# B&R Automation Studio project A2019059_Linka_Power_CP (part 43)

#### OvlServaZdvihu.st
```iecst
ACTION OvlServaZdvihu:

	//**************************Axis 11***********************************//
	//Otáčka serva = 10mm//
	//Motor má absolútny encodér a brzdu//

    //ENABLE knižnice//
    IF P4_Etiketovacka.ServoZdvihuEtiketovania_M28.STATUS.Communication_READY THEN
        P4_Etiketovacka.ServoZdvihuEtiketovania_M28.CMD.ENABLE:= TRUE;
    ELSE
        P4_Etiketovacka.ServoZdvihuEtiketovania_M28.CMD.ENABLE:= FALSE;
    END_IF

	//Zapnutie serva//
	CasPowerON.IN:= P4_Etiketovacka.ServoZdvihuEtiketovania_M28.STATUS.ReadyToPower_ON AND P4_Etiketovacka.STAV.ServoZvihu_LimitSnimace_BUSY AND P4_Etiketovacka.ServoZdvihuEtiketovania_M28.STATUS.EnableSwitch_ACTIVE AND NOT P4_Etiketovacka.ServoZdvihuEtiketovania_M28.STATUS.ERROR;
	IF CasPowerON.Q THEN
		P4_Etiketovacka.ServoZdvihuEtiketovania_M28.CMD.POWER:= TRUE;
	ELSE
		P4_Etiketovacka.ServoZdvihuEtiketovania_M28.CMD.POWER:= FALSE;
	END_IF

	CasPowerON.PT:= T#1s;
	CasPowerON();

    //Zobrazenie stavou a parametrov serva//
    P4_Etiketovacka.STAV.Zdvih_AktualnaPozicia:= P4_Etiketovacka.ServoZdvihuEtiketovania_M28.STATUS.ActualPosition;
	P4_Etiketovacka.STAV.Zdvih_AktualnaRychlost:= P4_Etiketovacka.ServoZdvihuEtiketovania_M28.STATUS.ActualVelocity;
	P4_Etiketovacka.STAV.Zdvih_AktualnyMoment:= P4_Etiketovacka.ServoZdvihuEtiketovania_M28.STATUS.ActualTorque;
	P4_Etiketovacka.STAV.ServoZdvihu_HomingOK:= P4_Etiketovacka.ServoZdvihuEtiketovania_M28.STATUS.Homing_OK;
	P4_Etiketovacka.STAV.ServoZdvihu_BUSY:= P4_Etiketovacka.ServoZdvihuEtiketovania_M28.STATUS.MoveAbsolute_BUSY;
	P4_Etiketovacka.STAV.Zdvih_JoggLimitDosiahnuty:= P4_Etiketovacka.ServoZdvihuEtiketovania_M28.STATUS.JoggLimit_Dosiahnuty;

	//Zadané parametre serva//
	P4_Etiketovacka.ServoZdvihuEtiketovania_M28.HomePAR.Acceleration:= 100;
	P4_Etiketovacka.ServoZdvihuEtiketovania_M28.HomePAR.HomingVelocity:= 5;
	P4_Etiketovacka.ServoZdvihuEtiketovania_M28.HomePAR.StartVelocity:= 10;
	P4_Etiketovacka.ServoZdvihuEtiketovania_M28.HomePAR.Position:= -21423.0;    //Offset homing pozície pre absolutny snímač
	P4_Etiketovacka.ServoZdvihuEtiketovania_M28.HomePAR.HomingMode:= 3; //0 - direct, 1- refrenčný snímač, 2 - limitný snímač, 3 - absolutny encoder, 4 - na moment//

	P4_Etiketovacka.ServoZdvihuEtiketovania_M28.PAR.Acceleration:= P34_RemPremenne.P4_ZdvihEtiketovacky_Rychlost*10;
	P4_Etiketovacka.ServoZdvihuEtiketovania_M28.PAR.Deceleration:= P34_RemPremenne.P4_ZdvihEtiketovacky_Rychlost*10;
	P4_Etiketovacka.ServoZdvihuEtiketovania_M28.PAR.StopDeceleration:= P34_RemPremenne.P4_ZdvihEtiketovacky_Rychlost*10;
	P4_Etiketovacka.ServoZdvihuEtiketovania_M28.PAR.Velocity:= P34_RemPremenne.P4_ZdvihEtiketovacky_Rychlost;
	P4_Etiketovacka.ServoZdvihuEtiketovania_M28.PAR.Position:= P4_Etiketovacka.PAR.ServoZdvihu_ZadanaPozicia;

	//Zastavenie pohybu serva//
	IF Zdvih_STOP THEN
		P4_Etiketovacka.ServoZdvihuEtiketovania_M28.CMD.STOP:= TRUE;
		SC_OvlZdvihu.Step:= 0;
		CasZastaveniaServa.IN:= TRUE;
		Zdvih_STOP:= FALSE;
	END_IF

	IF CasZastaveniaServa.Q THEN
		P4_Etiketovacka.ServoZdvihuEtiketovania_M28.CMD.STOP:= FALSE;
		CasZastaveniaServa.IN:= FALSE;
	END_IF

	CasZastaveniaServa.PT:= T#2s;
	CasZastaveniaServa();

	//Volanie funkcie SequenceControl//
	SequenceControl(SC:= SC_OvlZdvihu);

	CASE SC_OvlZdvihu.Step OF

		0:
			SC_OvlZdvihu.StepName:= '0 - Nulovanie';
			Zdvih_JoggHORE:= FALSE;
			Zdvih_JoggDOLE:= FALSE;
			Zdvih_POLOHUJ:= FALSE;
			Zdvih_HOME:= FALSE;
			P4_Etiketovacka.ServoZdvihuEtiketovania_M28.CMD.HOME:= FALSE;
			P4_Etiketovacka.ServoZdvihuEtiketovania_M28.CMD.JoggVPRED:= FALSE;
			P4_Etiketovacka.ServoZdvihuEtiketovania_M28.CMD.JoggVZAD:= FALSE;
			P4_Etiketovacka.ServoZdvihuEtiketovania_M28.CMD.MoveAbsolute:= FALSE;
			P4_Etiketovacka.ServoZdvihuEtiketovania_M28.CMD.MoveTorque:= FALSE;

			IF SC_P4_Etiketovacka.Step <> 0 AND P4_Etiketovacka.ServoZdvihuEtiketovania_M28.STATUS.Power_ON AND NOT P4_Etiketovacka.ServoZdvihuEtiketovania_M28.STATUS.ERROR AND NOT P4_Etiketovacka.ServoZdvihuEtiketovania_M28.STATUS.STOP_ACTIVE THEN
				SC_OvlZdvihu.ResetStep:= TRUE;
				SC_OvlZdvihu.Step:= 1;
			END_IF

		1:
			SC_OvlZdvihu.StepName:= '1 - Rozhodnutie o cinnosti';
			IF Zdvih_JoggHORE THEN
				SC_OvlZdvihu.Step:= 10;
			ELSIF Zdvih_JoggDOLE THEN
				SC_OvlZdvihu.Step:= 20;
			ELSIF Zdvih_HOME THEN
				SC_OvlZdvihu.Step:= 30;
			ELSIF Zdvih_POLOHUJ THEN
				SC_OvlZdvihu.Step:= 40;
			END_IF

		10:
			SC_OvlZdvihu.StepName:= '10 - Jogg HORE';
			SC_OvlZdvihu.IdleTime.PT:= T#3s;
			SC_OvlZdvihu.AlarmTime.PT:= T#3s;

			IF NOT SC_OvlZdvihu.Switch1 THEN
				P4_Etiketovacka.ServoZdvihuEtiketovania_M28.CMD.JoggVZAD:= TRUE;
				SC_OvlZdvihu.Switch1:= TRUE;
			END_IF

			IF NOT Zdvih_JoggHORE THEN
				SC_OvlZdvihu.ResetStep:= TRUE;
				SC_OvlZdvihu.Step:= 0;
			END_IF

		20:
			SC_OvlZdvihu.StepName:= '20 - Jogg DOLE';
			SC_OvlZdvihu.IdleTime.PT:= T#3s;
			SC_OvlZdvihu.AlarmTime.PT:= T#3s;

			IF NOT SC_OvlZdvihu.Switch1 THEN
				P4_Etiketovacka.ServoZdvihuEtiketovania_M28.CMD.JoggVPRED:= TRUE;
				SC_OvlZdvihu.Switch1:= TRUE;
			END_IF

			IF NOT Zdvih_JoggDOLE THEN
				SC_OvlZdvihu.ResetStep:= TRUE;
				SC_OvlZdvihu.Step:= 0;
			END_IF

		30:
			SC_OvlZdvihu.StepName:= '30 - Homing';
			SC_OvlZdvihu.IdleTime.PT:= T#500ms;
			SC_OvlZdvihu.AlarmTime.PT:= T#3s;

			IF NOT SC_OvlZdvihu.Switch1 THEN
				P4_Etiketovacka.ServoZdvihuEtiketovania_M28.CMD.HOME:= TRUE;
				SC_OvlZdvihu.IdleTime.IN:= TRUE;
				SC_OvlZdvihu.Switch1:= TRUE;
			END_IF

			IF P4_Etiketovacka.ServoZdvihuEtiketovania_M28.STATUS.Homing_OK AND SC_OvlZdvihu.IdleTime.Q THEN
				SC_OvlZdvihu.ResetStep:= TRUE;
				SC_OvlZdvihu.Step:= 0;
			END_IF

		40:
			SC_OvlZdvihu.StepName:= '40 - Polohovanie';
			SC_OvlZdvihu.IdleTime.PT:= T#500ms;
			SC_OvlZdvihu.AlarmTime.PT:= T#3s;

			ZadanaPoziciaUINT:= LREAL_TO_UINT(P4_Etiketovacka.PAR.ServoZdvihu_ZadanaPozicia);
			AktualnaPoziciaUINT:= LREAL_TO_UINT(P4_Etiketovacka.STAV.Zdvih_AktualnaPozicia);

			IF NOT SC_OvlZdvihu.Switch1 THEN
				P4_Etiketovacka.ServoZdvihuEtiketovania_M28.CMD.MoveAbsolute:= TRUE;
				SC_OvlZdvihu.Switch1:= TRUE;
			END_IF

			IF (AktualnaPoziciaUINT = ZadanaPoziciaUINT) AND P4_Etiketovacka.ServoZdvihuEtiketovania_M28.STATUS.MoveAbsolute_DONE THEN
				P4_Etiketovacka.STAV.ServoZdvihu_PoziciaDosiahnuta:= TRUE;
				SC_OvlZdvihu.ResetStep:= TRUE;
				SC_OvlZdvihu.Step:= 0;
			END_IF

	END_CASE

END_ACTION
```

#### KOM_Tlaciaren.st
```iecst
ACTION KOM_Tlaciaren:

	CASE Client.sStep OF

		0://Čakanie na spustenie komunikácie z tlačiarňou//
			IF Tlaciaren.Commands.VytlacEtiketu THEN
				Tlaciaren.Status.PoruchaOtvoreniaKomunikacie:= FALSE;
				Tlaciaren.Status.PoruchaSpojenia_s_Tlaciarnou:= FALSE;
				Tlaciaren.Status.PoruchaOdoslaniaDat:= FALSE;
				Tlaciaren.Status.PoruchaZatvoreniaKomunikacie:= FALSE;
				Tlaciaren.Status.PoruchaPrijatiaDat:= FALSE;
				Tlaciaren.Status.PrislaSprava_s_Tlaciarne:= FALSE;
				Tlaciaren.Status.VytlacenieEtikety_ERROR:= FALSE;
				(*strcpy(ADR(Tlaciaren.Data.Sprava_pre_Tlaciaren),ADR(''));*)
				strcpy(ADR(Tlaciaren.Data.Odpoved_s_Tlaciarne),ADR('')); //Vynulovanie premennej typu string
				Client.sStep := 1;
			END_IF

		1: //Otvorenie ethernetovej komunikácie//
			Client.TcpOpen_0.enable := 1;
			Client.TcpOpen_0.pIfAddr := 0;  (* Which Interface to open *)
			Client.TcpOpen_0.port := 9100;  (* Port komunikácie s tlačiarňou *)
			Client.TcpOpen_0.options := 0;
			Client.TcpOpen_0;  (* Call the Function *)

			IF Client.TcpOpen_0.status = 0 THEN  (* TCP port je otvorený *)
				Client.TcpOpen_timeout := 0;
				Client.sStep := 5;
			ELSIF Client.TcpOpen_0.status = ERR_FUB_BUSY THEN  (* TCP port sa otvára *)
				Client.TcpOpen_timeout := Client.TcpOpen_timeout + 1;
				IF Client.TcpOpen_timeout > 50 THEN
					Tlaciaren.Status.PoruchaOtvoreniaKomunikacie:= TRUE;
					Client.TcpOpen_timeout := 0;
					Client.sStep := 40;
				END_IF
				(* Busy *)
			ELSE  (* Goto Error Step *)
				Tlaciaren.Status.PoruchaOtvoreniaKomunikacie:= TRUE;
				Client.TcpOpen_timeout := 0;
				Tlaciaren.Status.VytlacenieEtikety_ERROR:= TRUE;
				Client.sStep := 100;
			END_IF

		5:
			Client.linger_opt.lLinger := 0; (* linger Time = 0 *)
			Client.linger_opt.lOnOff := 1; (* linger Option ON *)
			Client.TcpIoctl_0.enable := 1;
			Client.TcpIoctl_0.ident := Client.TcpOpen_0.ident; (* Connection Ident from AsTP.TCP_Open *)
			Client.TcpIoctl_0.ioctl := tcpSO_LINGER_SET; (* Set Linger Options *)
			Client.TcpIoctl_0.pData := ADR(Client.linger_opt);
			Client.TcpIoctl_0.datalen := SIZEOF(Client.linger_opt);
			Client.TcpIoctl_0;

			IF Client.TcpIoctl_0.status = 0 THEN  (* TcpIoctl successfull *)
				Client.sStep := 10;
			ELSIF Client.TcpIoctl_0.status = ERR_FUB_BUSY THEN  (* TcpIoctl not finished -> redo *)
				(* Busy *)
			ELSE  (* Goto Error Step *)
				Tlaciaren.Status.VytlacenieEtikety_ERROR:= TRUE;
				Client.sStep := 100;
			END_IF

		10: //Spojenie s tlačiarňou//
			Client.TcpClient_0.enable := 1;
			Client.TcpClient_0.ident := Client.TcpOpen_0.ident;  (* Connection Ident from AsTCP.TCP_Open *)
			Client.TcpClient_0.portserv := 9100;  (* Port komunikácie s tlačiarňou *)
			Client.TcpClient_0.pServer := ADR('192.168.122.41');  (* Adresa tlačiarne *)
			Client.TcpClient_0;  (* Call the Function*)

			IF Client.TcpClient_0.status = 0 THEN  (* Open ok -> Send Data *)
				Client.TcpClient_timeout := 0;
				Client.sStep := 20;
			ELSIF Client.TcpClient_0.status = ERR_FUB_BUSY THEN  (* TcpClient not finished -> redo *)
				Client.TcpClient_timeout := Client.TcpClient_timeout + 1;
				IF Client.TcpClient_timeout > 50 THEN
					Tlaciaren.Status.PoruchaSpojenia_s_Tlaciarnou:= TRUE;
					Client.TcpClient_timeout := 0;
					Client.sStep := 40;
				END_IF

				(* Busy *)
			ELSIF Client.TcpClient_0.status = tcpERR_INVALID THEN  (* Port error -> Close actual connection, and reopen a new one *)
				Client.TcpClient_timeout := 0;
				Client.sStep := 40;
			ELSE  (* Goto Error Step *)
				Tlaciaren.Status.PoruchaSpojenia_s_Tlaciarnou:= TRUE;
				Client.TcpClient_timeout := 0;
				Tlaciaren.Status.VytlacenieEtikety_ERROR:= TRUE;
				Client.sStep := 100;
			END_IF

		20: //Poslanie dát do tlačiarne//
			Client.TcpSend_0.enable := 1;
			Client.TcpSend_0.ident := Client.TcpOpen_0.ident;  (* Connection Ident from AsTCP.TCP_Open *)
			Client.TcpSend_0.pData := ADR(Tlaciaren.Data.Sprava_pre_Tlaciaren);  (* Dáta poslané do tlačiarne *)
			Client.TcpSend_0.datalen := SIZEOF(Tlaciaren.Data.Sprava_pre_Tlaciaren);  (* Lenght of data to send *)
			Client.TcpSend_0.flags := 0;
			Client.TcpSend_0;  (* Call the Function*)

			IF Client.TcpSend_0.status = 0 THEN  (* Data was sent sucessfully -> receive data *)
				Client.sStep := 40;
			ELSIF Client.TcpSend_0.status = ERR_FUB_BUSY THEN  (* TcpSend not finished -> redo *)
				(* Busy *)
			ELSIF (Client.TcpSend_0.status = tcpERR_SENTLEN) OR (Client.TcpSend_0.status = tcpERR_NOT_CONNECTED) THEN (* Connection Lost *)
				Client.sStep := 40;
			ELSE  (* Goto Error Step *)
				Tlaciaren.Status.PoruchaOdoslaniaDat:= TRUE;
				Tlaciaren.Status.VytlacenieEtikety_ERROR:= TRUE;
				Client.sStep := 100;
			END_IF

		30: //Prijatie odpovede s tlačiarne//
			Client.TcpRecv_0.enable := 1;
			Client.TcpRecv_0.ident := Client.TcpOpen_0.ident;  (* Connection Ident from AsTCP.TCP_Open *)
			Client.TcpRecv_0.pData	:= ADR(Tlaciaren.Data.Odpoved_s_Tlaciarne);  (* Dáta poslané z tlačiarne *)
			Client.TcpRecv_0.datamax := SIZEOF(Tlaciaren.Data.Odpoved_s_Tlaciarne);  (* Lenght of data buffer *)
			Client.TcpRecv_0.flags := 0;
			Client.TcpRecv_0;  (* Call the Function*)

			IF Client.TcpRecv_0.status = 0 THEN  (* Data was received sucessfully -> Send next packet *)
				Tlaciaren.Status.PrislaSprava_s_Tlaciarne:= TRUE;
				Client.recv_timeout := 0;
				Client.sStep := 40;
			ELSIF Client.TcpRecv_0.status = tcpERR_NO_DATA THEN  (* No data received - wait *)
				Client.recv_timeout := Client.recv_timeout + 1;
				IF Client.recv_timeout > 50 THEN
					Client.recv_timeout := 0;
					Client.sStep := 40;
				END_IF
				(* No Data received *)
			ELSIF Client.TcpRecv_0.status = ERR_FUB_BUSY THEN  (* TcpRecv not finished -> redo *)
				(* Busy *)
			ELSIF Client.TcpRecv_0.status = tcpERR_NOT_CONNECTED THEN (* Connection Lost *)
				Client.recv_timeout := 0;
				Client.sStep := 40;
			ELSE  (* Goto Error Step *)
				Tlaciaren.Status.PoruchaPrijatiaDat:= TRUE;
				Tlaciaren.Status.VytlacenieEtikety_ERROR:= TRUE;
				Client.recv_timeout := 0;
				Client.sStep := 100;
			END_IF

		40: //Zatvorenie ethernetovej komunikácie//
			Client.TcpClose_0.enable := 1;
			Client.TcpClose_0.ident := Client.TcpOpen_0.ident;  (* Connection Ident from AsTCP.TCP_Open *)
			Client.TcpClose_0.how := 0;
			Client.TcpClose_0;  (* Call the Function*)

			IF Client.TcpClose_0.status = 0 THEN  (* Close sucessfull -> Reopen the interface *)
				Tlaciaren.Status.VytlacenieEtikety_OK:= TRUE;
				Client.sStep := 100;
			ELSIF Client.TcpClose_0.status = ERR_FUB_BUSY THEN  (* TcpClose not finished -> redo *)
				(* Busy *)
			ELSE  (* Goto Error Step *)
				Tlaciaren.Status.PoruchaZatvoreniaKomunikacie:= TRUE;
				Tlaciaren.Status.VytlacenieEtikety_ERROR:= TRUE;
				Client.sStep := 100;
			END_IF

		100: //Ukončenie komunikácie s tlačiarňou//
			IF NOT Tlaciaren.Commands.VytlacEtiketu THEN
				Client.sStep := 0;
			END_IF

	END_CASE

END_ACTION
```

#### VytvorenieEtikety.st
```iecst
ACTION VytvorenieEtikety:

	//*********************************************Vyčítanie parametrov etikety zo servera*******************************************************//
	SerioveCisloEtikety;
	IF P4_Etiketovacka.RR_TestovanieEtiketovania THEN
		SerioveCisloEtikety:= 'T598454420120P32120001323091112';
	END_IF

	brsstrcpy(ADR(VstupnePoleUSINT),ADR(SerioveCisloEtikety)); //Skopirovanie vstupnej spravy do pola

    //***************************Vyčítanie Location Code*******************************************//
    brsmemcpy(ADR(Etiketa.LocationCode),ADR(VstupnePoleUSINT[1]),2);

    //**************************Vyčítanie Part Ident Number****************************************//
    brsmemcpy(ADR(Etiketa.PartIdentNumber),ADR(VstupnePoleUSINT[3]),7);

    //**************************Vyčítanie Change Index*********************************************//
    brsmemcpy(ADR(Etiketa.ChangeIndex),ADR(VstupnePoleUSINT[10]),2);

    //**************************Vyčítanie Production Year*********************************************//
    brsmemcpy(ADR(Etiketa.ProductionYear),ADR(VstupnePoleUSINT[12]),2);

    //**************************Vyčítanie Manufactured*********************************************//
    brsmemcpy(ADR(Etiketa.Manufactured),ADR(VstupnePoleUSINT[14]),1);

    //**************************Vyčítanie Day of production*********************************************//
    brsmemcpy(ADR(Etiketa.DayOfProduction),ADR(VstupnePoleUSINT[15]),3);

    //**************************Vyčítanie Assembly line*********************************************//
    brsmemcpy(ADR(Etiketa.AssemblyLine),ADR(VstupnePoleUSINT[18]),1);

    //**************************Vyčítanie Day production counter*********************************************//
    brsmemcpy(ADR(Etiketa.DayProductionCounter),ADR(VstupnePoleUSINT[19]),5);

    //**************************Vyčítanie Supplier number*********************************************//
    brsmemcpy(ADR(Etiketa.SuplierNumber),ADR(VstupnePoleUSINT[24]),6);

    //**************************Vyčítanie Supplier plant code*********************************************//
    brsmemcpy(ADR(Etiketa.PlantCode),ADR(VstupnePoleUSINT[30]),2);

    //*****************************************************Namapovanie parametrov etikety************************************************//

    //Identification number//
    EtiketaPanasonic.IdentificationNumber:= Etiketa.PartIdentNumber;

    //Change Index//
    EtiketaPanasonic.ChangeIndex:= '';
    strcat(ADR(EtiketaPanasonic.ChangeIndex),ADR('-'));
    strcat(ADR(EtiketaPanasonic.ChangeIndex),ADR(Etiketa.ChangeIndex));

    //Model type//
    EtiketaPanasonic.ModelType:= 'POWER-CP';

    //Supplier number//
	EtiketaPanasonic.SupplierNumber:= Etiketa.SuplierNumber;

    //Plant Code//
    EtiketaPanasonic.PlantCode:= Etiketa.PlantCode;

	//Country//
	EtiketaPanasonic.Country:= 'SK';

	//Dátum//
	EtiketaPanasonic.Date:= Den_STR;
	strcat(ADR(EtiketaPanasonic.Date),ADR('.'));
	strcat(ADR(EtiketaPanasonic.Date),ADR(Mesiac_STR));
	strcat(ADR(EtiketaPanasonic.Date),ADR('.'));
	strcat(ADR(EtiketaPanasonic.Date),ADR(Rok_STR_2_Znaky));

	//Counter//
	EtiketaPanasonic.Counter:= Etiketa.DayProductionCounter;

	//Data metrix kod//
	EtiketaPanasonic.DataMetrix:= SerioveCisloEtikety;

	//***************************************Správa pre tlačiareň Compa II*************************************************//
	Tlaciaren.Data.Sprava_pre_Tlaciaren:= '^XA';//Začiatok správy
	strcat(ADR(Tlaciaren.Data.Sprava_pre_Tlaciaren),ADR('^FO210,150^A8R,40,25^FD'));
	strcat(ADR(Tlaciaren.Data.Sprava_pre_Tlaciaren),ADR(EtiketaPanasonic.IdentificationNumber));
    strcat(ADR(Tlaciaren.Data.Sprava_pre_Tlaciaren),ADR('^FS'));
    strcat(ADR(Tlaciaren.Data.Sprava_pre_Tlaciaren),ADR('^FO210,274^A8R,40,25^FD'));
    strcat(ADR(Tlaciaren.Data.Sprava_pre_Tlaciaren),ADR(EtiketaPanasonic.ChangeIndex));
    strcat(ADR(Tlaciaren.Data.Sprava_pre_Tlaciaren),ADR('^FS'));
	strcat(ADR(Tlaciaren.Data.Sprava_pre_Tlaciaren),ADR('^FO172,188^A8R,40,25^FD'));
	strcat(ADR(Tlaciaren.Data.Sprava_pre_Tlaciaren),ADR(EtiketaPanasonic.ModelType));
	strcat(ADR(Tlaciaren.Data.Sprava_pre_Tlaciaren),ADR('^FS'));
	strcat(ADR(Tlaciaren.Data.Sprava_pre_Tlaciaren),ADR('^FO134,168^A8R,40,25^FD'));
	strcat(ADR(Tlaciaren.Data.Sprava_pre_Tlaciaren),ADR(EtiketaPanasonic.SupplierNumber));
    strcat(ADR(Tlaciaren.Data.Sprava_pre_Tlaciaren),ADR('^FS'));
    strcat(ADR(Tlaciaren.Data.Sprava_pre_Tlaciaren),ADR('^FO134,290^A8R,40,25^FD'));
    strcat(ADR(Tlaciaren.Data.Sprava_pre_Tlaciaren),ADR(EtiketaPanasonic.PlantCode));
    strcat(ADR(Tlaciaren.Data.Sprava_pre_Tlaciaren),ADR('^FS'));
	strcat(ADR(Tlaciaren.Data.Sprava_pre_Tlaciaren),ADR('^FO96,290^A8R,40,25^FD'));
	strcat(ADR(Tlaciaren.Data.Sprava_pre_Tlaciaren),ADR(EtiketaPanasonic.Country));
	strcat(ADR(Tlaciaren.Data.Sprava_pre_Tlaciaren),ADR('^FS'));
	strcat(ADR(Tlaciaren.Data.Sprava_pre_Tlaciaren),ADR('^FO58,185^A8R,40,25^FD'));
	strcat(ADR(Tlaciaren.Data.Sprava_pre_Tlaciaren),ADR(EtiketaPanasonic.Date));
	strcat(ADR(Tlaciaren.Data.Sprava_pre_Tlaciaren),ADR('^FS'));
	strcat(ADR(Tlaciaren.Data.Sprava_pre_Tlaciaren),ADR('^FO20,236^A8R,40,25^FD'));
	strcat(ADR(Tlaciaren.Data.Sprava_pre_Tlaciaren),ADR(EtiketaPanasonic.Counter));
	strcat(ADR(Tlaciaren.Data.Sprava_pre_Tlaciaren),ADR('^FS'));
	strcat(ADR(Tlaciaren.Data.Sprava_pre_Tlaciaren),ADR('^FO30,40^BXR,5,200^FD'));
	strcat(ADR(Tlaciaren.Data.Sprava_pre_Tlaciaren),ADR(EtiketaPanasonic.DataMetrix));
	strcat(ADR(Tlaciaren.Data.Sprava_pre_Tlaciaren),ADR('^FS'));
	strcat(ADR(Tlaciaren.Data.Sprava_pre_Tlaciaren),ADR('^XZ'));//Koniec správy

END_ACTION
```

### Program Logical/Program/Pracovisko_4/P4_OvladanieSafety (IEC)

#### Main.st - Init, cyclic, exit code
```iecst
PROGRAM _INIT
	(* Insert code here *)

END_PROGRAM

PROGRAM _CYCLIC

    //******************************************Ovládanie zámkov dverí bunky****************************************//
    //Predné dvere//
	IF EDGEPOS(P34_Vizu.TL_ZamkniPrednyZamok_P4) THEN
		IF NOT Safety.OUT.P4_ZamkniZamok_PredneDvere AND Safety.IN.P4_PredneDvere_PritomPetlice THEN
            Safety.OUT.P4_ZamkniZamok_PredneDvere:= TRUE;
        ELSIF Safety.OUT.P4_ZamkniZamok_PredneDvere THEN
            Safety.OUT.P4_ZamkniZamok_PredneDvere:= FALSE;
        END_IF
        P34_Vizu.TL_ZamkniPrednyZamok_P4:= FALSE;
    END_IF

    //Reset zóny bunky//
    CasResetZonyBunky.IN:= NOT Safety.STAV.P4_ZonaBunky_AKTIVNA	AND Safety.STAV.ZonaCS_AKTIVNA AND Safety.STAV.P4_ZamkyBunky_AKTIVNE AND (Safety.STAV.P4_VstupBunky_Bariera_AKTIVNA OR Safety.STAV.P4_VystupBunky_Bariera_AKTIVNA) AND (Safety.STAV.P3_VystupBunky_Bariera_AKTIVNA OR Safety.STAV.P3_ZamkyBunky_AKTIVNE);

	IF CasResetZonyBunky.Q THEN
		Safety.IN.P4_ZonaBunky_RESET:= TRUE;
	ELSE
		Safety.IN.P4_ZonaBunky_RESET:= FALSE;
	END_IF

	CasResetZonyBunky.PT:= T#1s;
	CasResetZonyBunky();

	//Reset zóny vytahu//
	CasResetZonyVytahu.IN:= NOT Safety.STAV.P4_ZonaVytahu_AKTIVNA AND Safety.STAV.ZonaCS_AKTIVNA AND (Safety.STAV.P4_Vytah_Bariera_AKTIVNA OR Safety.STAV.P4_SnimacVytahu_AKTIVNY);

	IF CasResetZonyVytahu.Q THEN
		Safety.IN.P4_ZonaVytahu_RESET:= TRUE;
	ELSE
		Safety.IN.P4_ZonaVytahu_RESET:= FALSE;
	END_IF

	CasResetZonyVytahu.PT:= T#1s;
	CasResetZonyVytahu();

END_PROGRAM

PROGRAM _EXIT
	(* Insert code here *)

END_PROGRAM
```

#### Variables.var - Local variables
```iecst
VAR
	CasResetZonyBunky : TON;
	CasResetZonyVytahu : TON;
END_VAR
```

### Program Logical/Program/Main (IEC)

#### Main.st - Init, cyclic, exit code
```iecst
PROGRAM _INIT
	(* Insert code here *)

END_PROGRAM

PROGRAM _CYCLIC

END_PROGRAM

PROGRAM _EXIT
	(* Insert code here *)

END_PROGRAM
```

- Visualisation Logical/mappView (not shown)

### Program Logical/Blikace/Blikanie100ms (IEC)

#### Blikanie100ms.st - Init, cyclic, exit code
```iecst
PROGRAM _INIT
	(* Insert code here *)

END_PROGRAM

PROGRAM _CYCLIC

	IF NOT Blikac100ms THEN
		Blikac100ms:= TRUE;
	ELSE
		Blikac100ms:= FALSE;
	END_IF

END_PROGRAM

PROGRAM _EXIT
	(* Insert code here *)

END_PROGRAM
```

### Program Logical/Blikace/Blikanie200ms (IEC)

#### Blikanie200ms.st - Init, cyclic, exit code
```iecst
PROGRAM _INIT
	(* Insert code here *)

END_PROGRAM

PROGRAM _CYCLIC

	IF NOT Blikac200ms THEN
		Blikac200ms:= TRUE;
	ELSE
		Blikac200ms:= FALSE;
	END_IF

END_PROGRAM

PROGRAM _EXIT
	(* Insert code here *)

END_PROGRAM
```

### Program Logical/Blikace/Blikanie500ms (IEC)

#### Blikanie500ms.st - Init, cyclic, exit code
```iecst
PROGRAM _INIT
	(* Insert code here *)

END_PROGRAM

PROGRAM _CYCLIC
	IF NOT Blikac500ms THEN
		Blikac500ms:= TRUE;
	ELSE
		Blikac500ms:= FALSE;
	END_IF

END_PROGRAM

PROGRAM _EXIT
	(* Insert code here *)

END_PROGRAM
```

### Program Logical/Blikace/Blikanie1s (IEC)

#### Blikanie1s.st - Init, cyclic, exit code
```iecst
PROGRAM _INIT
	(* Insert code here *)

END_PROGRAM

PROGRAM _CYCLIC
	IF NOT Blikac1s THEN
		Blikac1s:= TRUE;
	ELSE
		Blikac1s:= FALSE;
	END_IF

END_PROGRAM

PROGRAM _EXIT
	(* Insert code here *)

END_PROGRAM
```

### Program Logical/TracebilitySystem/P1_Vytah_ST1 (IEC)

#### Main.st - Init, cyclic, exit code
```iecst
PROGRAM _INIT

    SKTcpClientTrace_1.Params.IPportClient := 13000;
END_PROGRAM

PROGRAM _CYCLIC

//Priradenie indexu paletky//

    a:= P1_Vytah.PAR.IndexPaletky;

    //Parametre komunikácie//
    memcpy(ADR(SKTcpClientTrace_1.Params.IPaddrServ),ADR('192.168.122.250'),SIZEOF('192.168.122.250'));

    SKTcpClientTrace_1.Params.IPportServ := 12000;
    SKTcpClientTrace_1.Params.RecvTimeout := 10000;
    SKTcpClientTrace_1();

    //Parametre komunikácie//
    //Vstupy pre server//
    SKTcpClientTrace_1.Params.Packet.type := TRCB_P1_Vytah_ST1.INPUTS.TYP_Prikazu;
    SKTcpClientTrace_1.Params.Packet.workplace := TRCB_P1_Vytah_ST1.INPUTS.CisloStanice;
    TRCB_P1_Vytah_ST1.INPUTS.CisloPaletky:= 'Pal';
    brsstrcat(ADR(TRCB_P1_Vytah_ST1.INPUTS.CisloPaletky), ADR(P1_Vytah.PAR.IndexPaletky_STRING));
    SKTcpClientTrace_1.Params.Packet.rfid := TRCB_P1_Vytah_ST1.INPUTS.CisloPaletky;
    SKTcpClientTrace_1.Params.Packet.master := TRCB_P1_Vytah_ST1.INPUTS.QRkodPowerCP;
    SKTcpClientTrace_1.Params.Packet.dps1:= TRCB_P1_Vytah_ST1.INPUTS.QRkodFiltra;
    SKTcpClientTrace_1.Params.Packet.dps2:= '';
    SKTcpClientTrace_1.Params.Packet.dps3:= '';
    SKTcpClientTrace_1.Params.Packet.dps4:= '';
    SKTcpClientTrace_1.Params.Packet.dps5:= '';
    SKTcpClientTrace_1.Params.Packet.operator_id := TRCB_P1_Vytah_ST1.INPUTS.ID_Operatora;
    SKTcpClientTrace_1.Params.Packet.data_report:= TRCB_P1_Vytah_ST1.INPUTS.Report;
    SKTcpClientTrace_1.Params.Packet.result := TRCB_P1_Vytah_ST1.INPUTS.StavPaletky;

    ret := brsstrlen(ADR(TRCB_P1_Vytah_ST1.INPUTS.Report));

    //Výstupy zo servera//
    TRCB_P1_Vytah_ST1.OUTPUTS.TYP_Prikazu:= SKTcpClientTrace_1.Internal.Splitter.out[1];
    TRCB_P1_Vytah_ST1.OUTPUTS.CisloStanice:= SKTcpClientTrace_1.Internal.Splitter.out[2];
    TRCB_P1_Vytah_ST1.OUTPUTS.CisloPaletky:= SKTcpClientTrace_1.Internal.Splitter.out[3];
    IF TRCB_P1_Vytah_ST1.INPUTS.TYP_Prikazu = '0' THEN
        TRCB_P1_Vytah_ST1.OUTPUTS.CisloEtikety:= SKTcpClientTrace_1.Internal.Splitter.out[4];
    ELSE
        TRCB_P1_Vytah_ST1.OUTPUTS.QRkodPowerCP:= SKTcpClientTrace_1.Internal.Splitter.out[4];
    END_IF
    TRCB_P1_Vytah_ST1.OUTPUTS.QRkodFiltra:= SKTcpClientTrace_1.Internal.Splitter.out[5];
    TRCB_P1_Vytah_ST1.OUTPUTS.ID_Operatora:= SKTcpClientTrace_1.Internal.Splitter.out[10];
    TRCB_P1_Vytah_ST1.OUTPUTS.DruhCinnostiNaPaletke:= SKTcpClientTrace_1.Internal.Splitter.out[11];
    TRCB_P1_Vytah_ST1.OUTPUTS.PovolenieCinnostiNaPaletke:= SKTcpClientTrace_1.Internal.Splitter.out[12];

    //Volanie funkcie SequenceControl//
    SequenceControl(SC:= SC_KOM_Server);

    CASE SC_KOM_Server.Step OF

        0:
            SC_KOM_Server.StepName:= '0 - Nulovanie';
            SKTcpClientTrace_1.Cmd.Send:= FALSE;
            SKTcpClientTrace_1.Cmd.Close:= FALSE;
            TRCB_P1_Vytah_ST1.CMD.VyziadajStavPaletky_TYP1:= FALSE;
            TRCB_P1_Vytah_ST1.CMD.PriradQRkodFiltra_TYP3:= FALSE;
            TRCB_P1_Vytah_ST1.CMD.VyziadajCisloEtikety_TYP0:= FALSE;
            TRCB_P1_Vytah_ST1.CMD.OdosliStavPaletky_TYP2:= FALSE;
            TRCB_P1_Vytah_ST1.STATUS.KomunikaciaUkoncena:= FALSE;
            TRCB_P1_Vytah_ST1.STATUS.KomunikaciaError:= FALSE;
            PocetDopytovNaServer:= 0;

            IF SKTcpClientTrace_1.Internal.Step = 0 THEN
                SKTcpClientTrace_1.Enable:= TRUE;
                SC_KOM_Server.ResetStep:= TRUE;
                SC_KOM_Server.Step:= 1;
            ELSIF SKTcpClientTrace_1.Internal.Step = 15 THEN
                SKTcpClientTrace_1.Enable:= TRUE;
                SC_KOM_Server.ResetStep:= TRUE;
                SC_KOM_Server.Step:= 1;
            ELSE
                SKTcpClientTrace_1.Enable:= FALSE;
            END_IF

        1:
            SC_KOM_Server.StepName:= '1 - Rozhodnutie o cinnosti';
            IF TRCB_P1_Vytah_ST1.CMD.VyziadajStavPaletky_TYP1 THEN
                SC_KOM_Server.Step:= 10;
            ELSIF TRCB_P1_Vytah_ST1.CMD.PriradQRkodFiltra_TYP3 THEN
                SC_KOM_Server.Step:= 20;
            ELSIF TRCB_P1_Vytah_ST1.CMD.VyziadajCisloEtikety_TYP0 THEN
                SC_KOM_Server.Step:= 30;
            ELSIF TRCB_P1_Vytah_ST1.CMD.OdosliStavPaletky_TYP2 THEN
                SC_KOM_Server.Step:= 40;
            END_IF

        10:
            SC_KOM_Server.StepName:= '10 - Vyziadanie stavu paletky - odoslanie dat na server';
            SC_KOM_Server.IdleTime.PT:= T#3s;
            SC_KOM_Server.AlarmTime.PT:= T#10s;
            SC_KOM_Server.AlarmTime.IN:= TRUE;

            TRCB_P1_Vytah_ST1.INPUTS.TYP_Prikazu:= '1';
            TRCB_P1_Vytah_ST1.INPUTS.CisloStanice:= 'ST1';
            TRCB_P1_Vytah_ST1.INPUTS.CisloPaletky; //Z programu
            TRCB_P1_Vytah_ST1.INPUTS.QRkodPowerCP:= Paletka[a].PAR.QRkodPowerCP;
            TRCB_P1_Vytah_ST1.INPUTS.QRkodFiltra:= '';
            TRCB_P1_Vytah_ST1.INPUTS.ID_Operatora:= Paletka[a].PAR.ID_Operatora;
            TRCB_P1_Vytah_ST1.INPUTS.Report:= '';
            TRCB_P1_Vytah_ST1.INPUTS.StavPaletky:= 'OK';
            SKTcpClientTrace_1.Cmd.Send:= TRUE;

            IF SKTcpClientTrace_1.Cmd.Send AND NOT SKTcpClientTrace_1.Status.staReceived AND NOT SKTcpClientTrace_1.Status.staError THEN
                SC_KOM_Server.ResetStep:= TRUE;
                SC_KOM_Server.Step:= 13;
            ELSIF SC_KOM_Server.AlarmTime.Q AND (SKTcpClientTrace_1.Status.staReceived OR SKTcpClientTrace_1.Status.staError) THEN
                PocetDopytovNaServer:= PocetDopytovNaServer + 1;
                SKTcpClientTrace_1.Cmd.Send:= FALSE;
                SC_KOM_Server.ResetStep:= TRUE;
                SC_KOM_Server.Step:= 14;
            END_IF

        13:
            SC_KOM_Server.StepName:= '13 - Vyziadanie stavu paletky - odpoved servera';
            SC_KOM_Server.IdleTime.PT:= T#30s;
            SC_KOM_Server.AlarmTime.PT:= T#20s;
            SC_KOM_Server.AlarmTime.IN:= TRUE;

            IF SKTcpClientTrace_1.Status.staReceived AND
                (TRCB_P1_Vytah_ST1.OUTPUTS.TYP_Prikazu = TRCB_P1_Vytah_ST1.INPUTS.TYP_Prikazu) AND
                (TRCB_P1_Vytah_ST1.OUTPUTS.QRkodPowerCP = TRCB_P1_Vytah_ST1.INPUTS.QRkodPowerCP) THEN
                TRCB_P1_Vytah_ST1.STATUS.KomunikaciaUkoncena:= TRUE;
                SC_KOM_Server.ResetStep:= TRUE;
                SC_KOM_Server.Step:= 15;
            ELSIF SC_KOM_Server.AlarmTime.Q THEN
                PocetDopytovNaServer:= PocetDopytovNaServer + 1;
                SC_KOM_Server.ResetStep:= TRUE;
                SC_KOM_Server.Step:= 14;
            END_IF

        14:
            SC_KOM_Server.StepName:= '14 - Vyziadanie stavu paletky - cakam na opatovny dopyt na server';
            SC_KOM_Server.IdleTime.PT:= T#1s;
            SC_KOM_Server.AlarmTime.PT:= T#10s;
            SC_KOM_Server.IdleTime.IN:= TRUE;

            IF PocetDopytovNaServer < 3 THEN
                IF SC_KOM_Server.IdleTime.Q THEN
                    SC_KOM_Server.ResetStep:= TRUE;
                    SC_KOM_Server.Step:= 10;
                END_IF
            ELSE
                TRCB_P1_Vytah_ST1.STATUS.KomunikaciaError:= TRUE;
                SC_KOM_Server.ResetStep:= TRUE;
                SC_KOM_Server.Step:= 15;
            END_IF

        15:
            SC_KOM_Server.StepName:= '15 - Vyziadanie stavu paletky - cakam na ukoncenie komunikacie';
            SC_KOM_Server.IdleTime.PT:= T#3s;
            SC_KOM_Server.AlarmTime.PT:= T#10s;

            IF NOT TRCB_P1_Vytah_ST1.CMD.VyziadajStavPaletky_TYP1 THEN
                SC_KOM_Server.ResetStep:= TRUE;
                SC_KOM_Server.Step:= 0;
            END_IF

        20:
            SC_KOM_Server.StepName:= '20 - Priradenie QR kodu - odoslanie dat na server';
            SC_KOM_Server.IdleTime.PT:= T#3s;
            SC_KOM_Server.AlarmTime.PT:= T#5s;
            SC_KOM_Server.AlarmTime.IN:= TRUE;

            TRCB_P1_Vytah_ST1.INPUTS.TYP_Prikazu:= '3';
            TRCB_P1_Vytah_ST1.INPUTS.CisloStanice:= 'ST1';
            TRCB_P1_Vytah_ST1.INPUTS.CisloPaletky;
            TRCB_P1_Vytah_ST1.INPUTS.QRkodPowerCP:= Paletka[a].PAR.QRkodPowerCP;
            TRCB_P1_Vytah_ST1.INPUTS.QRkodFiltra:= Paletka[a].PAR.QRkodFiltra_4F5F;
            TRCB_P1_Vytah_ST1.INPUTS.ID_Operatora:= Paletka[a].PAR.ID_Operatora;
            TRCB_P1_Vytah_ST1.INPUTS.Report:= '';
            TRCB_P1_Vytah_ST1.INPUTS.StavPaletky:= 'OK';
            SKTcpClientTrace_1.Cmd.Send:= TRUE;

            IF SKTcpClientTrace_1.Cmd.Send AND NOT SKTcpClientTrace_1.Status.staReceived AND NOT SKTcpClientTrace_1.Status.staError THEN
                SC_KOM_Server.ResetStep:= TRUE;
                SC_KOM_Server.Step:= 23;
            ELSIF SC_KOM_Server.AlarmTime.Q AND (SKTcpClientTrace_1.Status.staReceived OR SKTcpClientTrace_1.Status.staError) THEN
                PocetDopytovNaServer:= PocetDopytovNaServer + 1;
                SC_KOM_Server.ResetStep:= TRUE;
                SC_KOM_Server.Step:= 24;
            END_IF

        23:
            SC_KOM_Server.StepName:= '23 - Priradenie QR kodu - odpoved servera';
            SC_KOM_Server.IdleTime.PT:= T#3s;
            SC_KOM_Server.AlarmTime.PT:= T#20s;
            SC_KOM_Server.AlarmTime.IN:= TRUE;

            IF SKTcpClientTrace_1.Status.staReceived AND
                (TRCB_P1_Vytah_ST1.OUTPUTS.TYP_Prikazu = TRCB_P1_Vytah_ST1.INPUTS.TYP_Prikazu) AND
                (TRCB_P1_Vytah_ST1.OUTPUTS.QRkodPowerCP = TRCB_P1_Vytah_ST1.INPUTS.QRkodPowerCP) THEN
                TRCB_P1_Vytah_ST1.STATUS.KomunikaciaUkoncena:= TRUE;
                SC_KOM_Server.ResetStep:= TRUE;
                SC_KOM_Server.Step:= 25;
            ELSIF SC_KOM_Server.AlarmTime.Q THEN
                PocetDopytovNaServer:= PocetDopytovNaServer + 1;
                SC_KOM_Server.ResetStep:= TRUE;
                SC_KOM_Server.Step:= 24;
            END_IF

        24:
            SC_KOM_Server.StepName:= '24 - Priradenie QR kodu - cakam na opatovny dopyt na server';
            SC_KOM_Server.IdleTime.PT:= T#1s;
            SC_KOM_Server.AlarmTime.PT:= T#10s;
            SC_KOM_Server.IdleTime.IN:= TRUE;
            SKTcpClientTrace_1.Cmd.Send:= FALSE;

            IF PocetDopytovNaServer < 3 THEN
                IF SC_KOM_Server.IdleTime.Q THEN
                    SC_KOM_Server.ResetStep:= TRUE;
                    SC_KOM_Server.Step:= 20;
                END_IF
            ELSE
                TRCB_P1_Vytah_ST1.STATUS.KomunikaciaError:= TRUE;
                SC_KOM_Server.ResetStep:= TRUE;
                SC_KOM_Server.Step:= 25;
            END_IF

        25:
            SC_KOM_Server.StepName:= '25 - Vyziadanie stavu paletky - cakam na ukoncenie komunikacie';
            SC_KOM_Server.IdleTime.PT:= T#3s;
            SC_KOM_Server.AlarmTime.PT:= T#10s;

            IF NOT TRCB_P1_Vytah_ST1.CMD.PriradQRkodFiltra_TYP3 THEN
                SC_KOM_Server.ResetStep:= TRUE;
                SC_KOM_Server.Step:= 0;
            END_IF

        30:
            SC_KOM_Server.StepName:= '30 - Vyziadanie serioveho cisla - odoslanie dat na server';
            SC_KOM_Server.IdleTime.PT:= T#3s;
            SC_KOM_Server.AlarmTime.PT:= T#10s;

            TRCB_P1_Vytah_ST1.INPUTS.TYP_Prikazu:= '0';
            TRCB_P1_Vytah_ST1.INPUTS.CisloStanice:= 'ST1';
            TRCB_P1_Vytah_ST1.INPUTS.CisloPaletky;
            TRCB_P1_Vytah_ST1.INPUTS.QRkodPowerCP:= '';
            TRCB_P1_Vytah_ST1.INPUTS.QRkodFiltra:= '';
            TRCB_P1_Vytah_ST1.INPUTS.ID_Operatora:= 'E2';
            TRCB_P1_Vytah_ST1.INPUTS.Report:= '';
            TRCB_P1_Vytah_ST1.INPUTS.StavPaletky:= 'OK';
            SKTcpClientTrace_1.Cmd.Send:= TRUE;

            IF SKTcpClientTrace_1.Cmd.Send AND NOT SKTcpClientTrace_1.Status.staReceived AND NOT SKTcpClientTrace_1.Status.staError THEN
                SC_KOM_Server.ResetStep:= TRUE;
                SC_KOM_Server.Step:= 33;
            END_IF

        33:
            SC_KOM_Server.StepName:= '33 - Vyziadanie serioveho cisla - odpoved servera';
            SC_KOM_Server.IdleTime.PT:= T#3s;
            SC_KOM_Server.AlarmTime.PT:= T#20s;
            SC_KOM_Server.AlarmTime.IN:= TRUE;

            IF SKTcpClientTrace_1.Status.staReceived AND
                (TRCB_P1_Vytah_ST1.OUTPUTS.TYP_Prikazu = TRCB_P1_Vytah_ST1.INPUTS.TYP_Prikazu) THEN
                TRCB_P1_Vytah_ST1.STATUS.KomunikaciaUkoncena:= TRUE;
                SC_KOM_Server.ResetStep:= TRUE;
                SC_KOM_Server.Step:= 35;
            ELSIF SC_KOM_Server.AlarmTime.Q THEN
                TRCB_P1_Vytah_ST1.STATUS.KomunikaciaError:= TRUE;
                SC_KOM_Server.ResetStep:= TRUE;
                SC_KOM_Server.Step:= 35;
            END_IF

        35:
            SC_KOM_Server.StepName:= '35 - Vyziadanie serioveho cisla - cakam na ukoncenie komunikacie';
            SC_KOM_Server.IdleTime.PT:= T#3s;
            SC_KOM_Server.AlarmTime.PT:= T#10s;

            IF NOT TRCB_P1_Vytah_ST1.CMD.VyziadajCisloEtikety_TYP0 THEN
                SC_KOM_Server.ResetStep:= TRUE;
                SC_KOM_Server.Step:= 0;
            END_IF

        40:
            SC_KOM_Server.StepName:= '40 - Odoslanie stavu paletky - odoslanie dat na server';
            SC_KOM_Server.IdleTime.PT:= T#3s;
            SC_KOM_Server.AlarmTime.PT:= T#20s;
            SC_KOM_Server.AlarmTime.IN:= TRUE;

            //Vytvorenie spravy pre report//

            IF NOT SC_KOM_Server.Switch1 THEN
				brsmemset(ADR(Report),0,SIZEOF(Report));
				brsmemset(ADR(TRCB_P1_Vytah_ST1.INPUTS.Report), 0, SIZEOF(TRCB_P1_Vytah_ST1.INPUTS.Report));

                //Kamera 2 - Kontrola paletky//
                Report[0].PoradoveCislo:= '1';
                Report[0].Popis:= 'KAM_2_KontrolaPaletky';
                Report[0].FormatHodnoty:= '2';
                Report[0].Tolerancia_MIN_Hodnota:= '';
                Report[0].Tolerancia_MAX_Hodnota:= '';
                Report[0].Nominal:= 'OK';
                Report[0].Tolerancia_MIN_Jednotky:= '';
                Report[0].Tolerancia_MAX_Jednotky:= '';
                IF Reports.Kamery.P1_CAM2_KontrolaPaletky = 'PASS' THEN
                    Report[0].NameranaHodnota:= 'OK';
                ELSE
                    Report[0].NameranaHodnota:= 'NG';
                END_IF
                Report[0].NameranaHodnota_Jednotky:= '';
                Report[0].VyslednyResult:= Reports.Kamery.P1_CAM2_KontrolaPaletky;
                SKTcpClientNewCsvEntry(Report[0].PoradoveCislo,Report[0].Popis,Report[0].FormatHodnoty,Report[0].Tolerancia_MIN_Hodnota,Report[0].Tolerancia_MAX_Hodnota,Report[0].Nominal,Report[0].Tolerancia_MIN_Jednotky,Report[0].Tolerancia_MAX_Jednotky,Report[0].NameranaHodnota,Report[0].NameranaHodnota_Jednotky,Report[0].VyslednyResult, ADR(TRCB_P1_Vytah_ST1.INPUTS.Report));

                //Kamera 4 - Kontrola pinov DPS//
                Report[1].PoradoveCislo:= '2';
                Report[1].Popis:= 'KAM_4_KontrolaPinovDPS';
                Report[1].FormatHodnoty:= '2';
                Report[1].Tolerancia_MIN_Hodnota:= '';
                Report[1].Tolerancia_MAX_Hodnota:= '';
                Report[1].Nominal:= 'OK';
                Report[1].Tolerancia_MIN_Jednotky:= '';
                Report[1].Tolerancia_MAX_Jednotky:= '';
                IF Reports.Kamery.P1_CAM4_KontrolaPinovDPS = 'PASS' THEN
                    Report[1].NameranaHodnota:= 'OK';
                ELSE
                    Report[1].NameranaHodnota:= 'NG';
                END_IF
                Report[1].NameranaHodnota_Jednotky:= '';
                Report[1].VyslednyResult:= Reports.Kamery.P1_CAM4_KontrolaPinovDPS;
                SKTcpClientNewCsvEntry(Report[1].PoradoveCislo,Report[1].Popis,Report[1].FormatHodnoty,Report[1].Tolerancia_MIN_Hodnota,Report[1].Tolerancia_MAX_Hodnota,Report[1].Nominal,Report[1].Tolerancia_MIN_Jednotky,Report[1].Tolerancia_MAX_Jednotky,Report[1].NameranaHodnota,Report[1].NameranaHodnota_Jednotky,Report[1].VyslednyResult, ADR(TRCB_P1_Vytah_ST1.INPUTS.Report));

                SC_KOM_Server.Switch1:= TRUE;
            END_IF

            TRCB_P1_Vytah_ST1.INPUTS.TYP_Prikazu:= '2';
            TRCB_P1_Vytah_ST1.INPUTS.CisloStanice:= 'ST1';
            TRCB_P1_Vytah_ST1.INPUTS.CisloPaletky;
            TRCB_P1_Vytah_ST1.INPUTS.QRkodPowerCP:= Paletka[a].PAR.QRkodPowerCP;
            TRCB_P1_Vytah_ST1.INPUTS.QRkodFiltra:= '';
            TRCB_P1_Vytah_ST1.INPUTS.ID_Operatora:= Paletka[a].PAR.ID_Operatora;;
            TRCB_P1_Vytah_ST1.INPUTS.StavPaletky:= Paletka[a].PAR.StavPowerCP;
            SKTcpClientTrace_1.Cmd.Send:= TRUE;

            IF SKTcpClientTrace_1.Cmd.Send AND NOT SKTcpClientTrace_1.Status.staReceived AND NOT SKTcpClientTrace_1.Status.staError THEN
                SC_KOM_Server.ResetStep:= TRUE;
                SC_KOM_Server.Step:= 43;
            ELSIF SC_KOM_Server.AlarmTime.Q AND (SKTcpClientTrace_1.Status.staReceived OR SKTcpClientTrace_1.Status.staError) THEN
                PocetDopytovNaServer:= PocetDopytovNaServer + 1;
                SC_KOM_Server.ResetStep:= TRUE;
                SC_KOM_Server.Step:= 44;
            END_IF

        43:
            SC_KOM_Server.StepName:= '43 - Odoslanie stavu paletky - odpoved servera';
            SC_KOM_Server.IdleTime.PT:= T#3s;
            SC_KOM_Server.AlarmTime.PT:= T#20s;
            SC_KOM_Server.AlarmTime.IN:= TRUE;

            IF SKTcpClientTrace_1.Status.staReceived AND
                (TRCB_P1_Vytah_ST1.OUTPUTS.TYP_Prikazu = TRCB_P1_Vytah_ST1.INPUTS.TYP_Prikazu) AND
                (TRCB_P1_Vytah_ST1.OUTPUTS.QRkodPowerCP = TRCB_P1_Vytah_ST1.INPUTS.QRkodPowerCP) THEN
                TRCB_P1_Vytah_ST1.STATUS.KomunikaciaUkoncena:= TRUE;
                SC_KOM_Server.ResetStep:= TRUE;
                SC_KOM_Server.Step:= 45;
            ELSIF SC_KOM_Server.AlarmTime.Q THEN
                PocetDopytovNaServer:= PocetDopytovNaServer + 1;
                SC_KOM_Server.ResetStep:= TRUE;
                SC_KOM_Server.Step:= 44;
            END_IF

        44:
            SC_KOM_Server.StepName:= '44 - Odoslanie stavu paletky - cakam na opatovny dopyt na server';
            SC_KOM_Server.IdleTime.PT:= T#1s;
            SC_KOM_Server.AlarmTime.PT:= T#10s;
            SC_KOM_Server.IdleTime.IN:= TRUE;
            SKTcpClientTrace_1.Cmd.Send:= FALSE;

            IF PocetDopytovNaServer < 3 THEN
                IF SC_KOM_Server.IdleTime.Q THEN
                    SC_KOM_Server.ResetStep:= TRUE;
                    SC_KOM_Server.Step:= 40;
                END_IF
            ELSE
                TRCB_P1_Vytah_ST1.STATUS.KomunikaciaError:= TRUE;
                SC_KOM_Server.ResetStep:= TRUE;
                SC_KOM_Server.Step:= 45;
            END_IF

        45:
            SC_KOM_Server.StepName:= '45 - Odoslanie stavu paletky - cakam na ukoncenie komunikacie';
            SC_KOM_Server.IdleTime.PT:= T#3s;
            SC_KOM_Server.AlarmTime.PT:= T#10s;

            IF NOT TRCB_P1_Vytah_ST1.CMD.OdosliStavPaletky_TYP2 THEN
                SC_KOM_Server.ResetStep:= TRUE;
                SC_KOM_Server.Step:= 0;
            END_IF

    END_CASE

            END_PROGRAM

PROGRAM _EXIT
            (* Insert code here *)

            END_PROGRAM
```

#### Types.typ - Local data types
```iecst
TYPE
	Report_typ : 	STRUCT
		PoradoveCislo : STRING[2]; (*IDstep - Poradové čislo reportu*)
		Popis : STRING[100]; (*Description - Popis*)
		FormatHodnoty : STRING[2]; (*TypValue - Format zaslané hodnoty  1- Číslo, 2 - Znak*)
		Tolerancia_MIN_Hodnota : STRING[10]; (*MinTol - Minimálna tolerancia meranej veličiny*)
		Tolerancia_MAX_Hodnota : STRING[10]; (*MaxTol - Maximálna tolerancia meranej veličiny*)
		Nominal : STRING[10]; (*Nom - Ak jezvolený formát string tak tu zadáme OK inak je prazdna*)
		Tolerancia_MIN_Jednotky : STRING[10]; (*MinEle - Jednotky minimálnej tolerancie veličiny*)
		Tolerancia_MAX_Jednotky : STRING[10]; (*MaxEle - Jednotky maximálnej tolerancie veličiny*)
		NameranaHodnota : STRING[10]; (*Value - Namerana hodnota veličiny, ak su kamery tak bude hodnota OK alebo NG*)
		NameranaHodnota_Jednotky : STRING[10]; (*ValEle - Jednotky nameranej veličiny*)
		VyslednyResult : STRING[5]; (*Result - Výsledný result  PASS, FAIL, SKIP*)
	END_STRUCT;
END_TYPE
```

#### Variables.var - Local variables
```iecst
VAR
	SC_KOM_Server : SequenceControlTyp;
	SKTcpClientTrace_1 : SKTcpClientTrace;
	a : USINT;
	Report : ARRAY[0..50] OF Report_typ;
	ret : UDINT;
	PocetDopytovNaServer : USINT;
END_VAR
```

### Program Logical/TracebilitySystem/P1_Srobovanie_ST2 (IEC)
